{attribute 'GeneratedUsingTerminal: EP6228-3132-0016'}
{attribute addProperty BoxType "EP6228-3132-0016"}
{attribute addProperty Id "Pin2_Ch1AT %I*BOOL1Pin2_Ch2AT %I*BOOL1Pin2_Ch5AT %I*BOOL1Pin2_Ch6AT %I*BOOL1"}
{attribute addProperty CRC "1038888231"}
{attribute addProperty Size "4"}
TYPE Digital_Inputs_3DEC2D27 EXTENDS InputBase_8311D824 :
STRUCT
	{attribute addProperty Name "Pin2_Ch1"}
	Pin2_Ch1 AT %I* : BOOL;
	{attribute addProperty Name "Pin2_Ch2"}
	Pin2_Ch2 AT %I* : BOOL;
	{attribute addProperty Name "Pin2_Ch5"}
	Pin2_Ch5 AT %I* : BOOL;
	{attribute addProperty Name "Pin2_Ch6"}
	Pin2_Ch6 AT %I* : BOOL;
END_STRUCT
END_TYPE

(* stored: Version 1.2.0.0, ProductVersion 3.1.4024.9
   DUT Digital_Inputs_3DEC2D27: Id {166519ac-574d-4fa4-b6eb-3dd03e9fef12} *)
